FUNCTION_BLOCK FB_CONTROL_SET2 (* Basic Function Block Type *)
  (* Standard: 61499-2 *)
  (* Version 0.0, 2011-08-24, 4DIAC-IDE, 4DIAC-Consortium *)
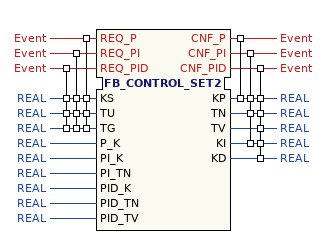
  EVENT_INPUT
    REQ_P WITH KS, TU, TG; (* request calcuation for P *)
    REQ_PI WITH KS, TU, TG; (* request calculation for PI *)
    REQ_PID WITH KS, TU, TG; (* request calculation for PID *)
  END_EVENT
  EVENT_OUTPUT
    CNF_P WITH KP; (* Execution Confirmation *)
    CNF_PI WITH KP, TN, KI;
    CNF_PID WITH KP, TN, TV, KI, KD;
  END_EVENT
  VAR_INPUT
    KS : REAL; (* critical gain *)
    TU : REAL;
    TG : REAL;
    P_K : REAL := 1.0; (* default value KP for P controller *)
    PI_K : REAL := 0.9; (* default value KP for PI controller *)
    PI_TN : REAL := 3.33; (* default value TN for PI controller *)
    PID_K : REAL := 1.2; (* default value KP for PID controller *)
    PID_TN : REAL := 2.0; (* default value TN for PID controller *)
    PID_TV : REAL := 0.5; (* default value TV for PID controller *)
  END_VAR
  VAR_OUTPUT
    KP : REAL; (* variable gain *)
    TN : REAL; (* past set time of the integrator *)
    TV : REAL; (* retention time of the differentiator *)
    KI : REAL; (* gain of the integrator *)
    KD : REAL; (* gain of the differentiator *)
  END_VAR
  VAR
    TX : REAL;
  END_VAR
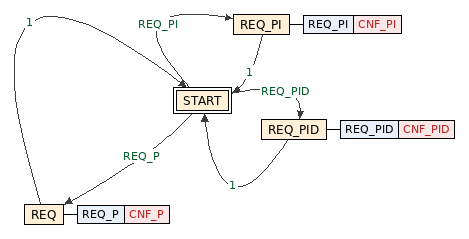
  EC_STATES
    START; (* Initial State *)
    REQ : REQ_P -> CNF_P; (* Normal execution *)
    REQ_PI : REQ_PI -> CNF_PI;
    REQ_PID : REQ_PID -> CNF_PID;
  END_STATES
  EC_TRANSITIONS
    START TO REQ := REQ_P;
    REQ TO START := 1;
    START TO REQ_PI := REQ_PI;
    REQ_PI TO START := 1;
    START TO REQ_PID := REQ_PID;
    REQ_PID TO START := 1;
  END_TRANSITIONS
  ALGORITHM REQ_P IN ST: (* Normally executed algorithm *)
(* Testing new idea planed for IEC61499-5 that allows to call other algs *)
CALC_TX();

KP := P_K * TX;
  END_ALGORITHM
  ALGORITHM REQ_PI IN ST: (* ALG *)
(* Testing new idea planed for IEC61499-5 that allows to call other algs *)
CALC_TX();

KP := PI_K * TX;
TN := PI_TN * TU;

CALC_KI();
  END_ALGORITHM
  ALGORITHM REQ_PID IN ST: (* ALG *)
(* Testing new idea planed for IEC61499-5 that allows to call other algs *)
CALC_TX();

KP := PID_K * TX;
TN := PID_TN * TU;
TV := PID_TV * TU;

CALC_KI();

KD := KP * TV;
  END_ALGORITHM
  ALGORITHM CALC_TX IN ST: (* ALG *)
TX := 0.0;
IF TU > 0.0 AND KS > 0.0 THEN TX := TG / TU / KS; END_IF;
  END_ALGORITHM
  ALGORITHM CALC_KI IN ST: (* ALG *)
IF TN > 0.0 THEN KI := KP / TN; ELSE KI := 0.0; END_IF;
  END_ALGORITHM
END_FUNCTION_BLOCK
